# EPICS substitutions: RKNPS/RKNPS-IOC-01App/Db/riken_rb2_mode_changeover_psus.substitutions
file riken_psus.template {
#
# PSNAME = Name of the IOC. e.g. "RB1", "RB2"
# PSIOC  = IOC which this power supply is on. E.g. RKNPS_01
# PSIDX  = Letter A-L. Must be unique
#
pattern {PV_PREFIX, P, PSU_DISABLE, PSNAME, PSIOC, PSIDX}

    {"\$(PV_PREFIX)", "\$(P)", "\$(PSU_DISABLE)", "RB2", "RKNPS_01", "A"}
    {"\$(PV_PREFIX)", "\$(P)", "\$(PSU_DISABLE)", "RB2-2", "RKNPS_01", "B"}
}
